{attribute 'qualified_only'}
TYPE E_State :
(
	Init := 0,
	ReadOnce,
	ReadPeriodically,
	Error,
	
	Idle,
	DeleteFolder,
	ReadOnce_CpuUsage,
	ReadOnce_CpuTemperature,
	ReadOnce_SrnMainboard,
	ReadOnce_SrnIPC,
	ReadBios,
	Write_DHCP,
	Write_IPAddr,
	SetAmsNetId
);
END_TYPE

(* stored: Version 1.1.0.1, ProductVersion 3.1.4024.12
   DUT E_State: Id {152610e0-cdbf-4e25-93df-dac94cd9b39b} *)
